(* CoDeSys 2.3.9.37 project: CapB_4.pro *)
(* Libraries: Standard.lib 4.10.05 12:14:46, IecSfc.lib 13.4.06 16:51:28, SYSLIBCALLBACK.LIB 26.9.08 17:43:52 *)

(* POU PLC_PRG, ST *)
PROGRAM PLC_PRG
VAR
     SeleccionX:INT:=1;
     SeleccionY:INT:=1;
      Tabla: ARRAY [1..10,1..20] OF INT;
	i: INT;
	j: INT;
	Duplica: BOOL;
END_VAR
FOR i:=1 TO 10 DO
   FOR j:=1 TO 20 DO
      IF Duplica THEN
         Tabla[i,j]:=2*i*j;
      ELSE
         Tabla[i,j]:=i*j;
     END_IF
   END_FOR
END_FOR
END_PROGRAM

(* Visualisation EjemploVisu
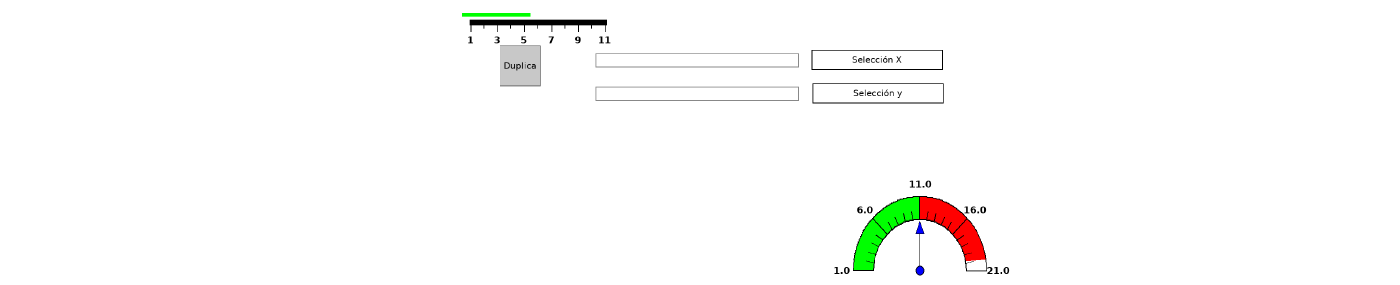
button at (45,38)-(92,85): text "Duplica"; toggles PLC_PRG.Duplica
rectangle at (407,43)-(559,66): text "Selección X"
rectangle at (408,82)-(560,105): text "Selección y"
group at (428,184)-(638,309)
  rectangle at (0,0)-(1,1): text "{ExtendedElement},Visu\ElementDLL.ete,0,@Zeigerinstrument,210,180,0,0,0,0,255,0,PLC_PRG.SeleccionY,,%.1f,0,1,1,1,5,1,21,0,0,0,0,0,0,0,-13,16,700,Arial,1,2,1,11,0,255,0,11,20,255,0,0,0,255,255,255,,0,0,0,0,"
  rectangle at (3,97)-(25,113): text "1.0"
  rectangle at (30,33)-(52,49): text "6.0"
  rectangle at (91,6)-(120,22): text "11.0"
  rectangle at (155,33)-(184,49): text "16.0"
  rectangle at (182,97)-(211,113): text "21.0"
  polygon at (100,53)-(110,105): angle ((PLC_PRG.SeleccionY * 1.0)-11) * 9
rectangle at (0,0)-(1,1): text "{ExtendedElement},Visu\ElementDLL.ete,1,@Bargraph,179,49,0,0,0,PLC_PRG.SeleccionX,,%1.0f,1,2,1,11,0,0,0,0,0,0,0,-13,16,700,Arial,0,255,0,255,0,0,0,0,1,0,0,1,0,,0,0,0,"
rectangle at (1,0)-(80,4): alarm colour if (PLC_PRG.SeleccionX) < 0; right ((PLC_PRG.SeleccionX * 1.0) - 6)  * 15.6
rectangle at (6,24)-(15,45): text "1"
rectangle at (37,24)-(46,45): text "3"
rectangle at (68,24)-(77,45): text "5"
rectangle at (100,24)-(109,45): text "7"
rectangle at (131,24)-(140,45): text "9"
rectangle at (157,24)-(176,45): text "11"
41 more shapes without text or variables
*)
